FUNCTION_BLOCK Test_NotificationNoArgs EXTENDS T_UnitTestBase
VAR
    Notification        : T_Notification;
    NotificationHandler : T_NotificationHandler;
    IsRaised            : BOOL;
    Assertion           : T_Assertion;
END_VAR

{attribute 'analysis' := '-33'} // inhibit unused variable warning
METHOD RunTest
VAR_OUTPUT
    TestCompleted : BOOL;
    TestFailed    : BOOL;
END_VAR
NotificationHandler.FB_init(bInitRetains    := FALSE,
                            bInCopyCode     := FALSE);

Notification.ClearNotificationHandlers().AddNotificationHandler(NotificationHandler);

Notification.Raise();
IsRaised := NotificationHandler.IsRaised();

TestFailed S= NOT Assertion.AssertEquals_BOOL(Source       := TestName,
                                              Expected     := TRUE,
                                              Actual       := IsRaised,
                                              VariableName := 'IsRaised');

TestCompleted := TRUE;
END_METHOD

END_FUNCTION_BLOCK

(* stored: Version 1.1.0.1, ProductVersion 3.1.4024.12
   POU Test_NotificationNoArgs: Id {b0e0872e-d94f-4d7d-8638-6a5be13a36bd}, SpecialFunc None
   Method RunTest: Id {05a006be-4cb6-4ddd-80b2-0abb8e5d388d} *)
